// TIA Portal V20 export
FUNCTION "Program" : Void   // FC1, LAD
{ S7_Optimized_Access := 'TRUE' }
// stored: SetENOAutomatically false
BEGIN

REGION Network 1
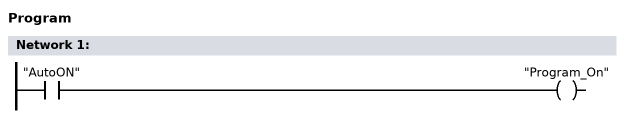
   RUNG wire#powerrail
      Contact( "AutoON" )
      Coil( "Program_On" )
   END_RUNG
   // the same network as SCL:
   "Program_On" := "AutoON";
END_REGION
END_FUNCTION
